// TIA Portal V21 program export: 3 tag tables, 4 data types, 7 data blocks, 12 code blocks (in call order from the OBs), 2 instance data blocks

VAR_GLOBAL   // PLC tag table "DIAG"
   D_Supply_MOD2 AT %I200.0 : Bool;   //    {ExternalWritable false}
   D_Supply_MOD3 AT %I200.1 : Bool;   //    {ExternalWritable false}
   D_Supply_MOD4 AT %I200.2 : Bool;   //    {ExternalWritable false}
   D_Supply_MOD5 AT %I200.3 : Bool;   //    {ExternalWritable false}
   D_Reserve_200_4 AT %I200.4 : Bool;   //    {ExternalWritable false}
   D_Reserve_200_5 AT %I200.5 : Bool;   //    {ExternalWritable false}
   D_Reserve_200_6 AT %I200.6 : Bool;   //    {ExternalWritable false}
   D_Reserve_200_7 AT %I200.7 : Bool;   //    {ExternalWritable false}
   D_Reserve_201_0 AT %I201.0 : Bool;   //    {ExternalWritable false}
   D_Reserve_201_1 AT %I201.1 : Bool;   //    {ExternalWritable false}
   D_Reserve_201_2 AT %I201.2 : Bool;   //    {ExternalWritable false}
   D_Reserve_201_3 AT %I201.3 : Bool;   //    {ExternalWritable false}
   D_Reserve_201_4 AT %I201.4 : Bool;   //    {ExternalWritable false}
   D_Reserve_201_5 AT %I201.5 : Bool;   //    {ExternalWritable false}
   D_Reserve_201_6 AT %I201.6 : Bool;   //    {ExternalWritable false}
   D_Reserve_201_7 AT %I201.7 : Bool;   //    {ExternalWritable false}
   D_Reserve_202_0 AT %I202.0 : Bool;   //    {ExternalWritable false}
   D_Reserve_202_1 AT %I202.1 : Bool;   //    {ExternalWritable false}
   D_Reserve_202_2 AT %I202.2 : Bool;   //    {ExternalWritable false}
   D_Reserve_202_3 AT %I202.3 : Bool;   //    {ExternalWritable false}
   D_Reserve_202_4 AT %I202.4 : Bool;   //    {ExternalWritable false}
   D_Reserve_202_5 AT %I202.5 : Bool;   //    {ExternalWritable false}
   D_Reserve_202_6 AT %I202.6 : Bool;   //    {ExternalWritable false}
   D_Reserve_202_7 AT %I202.7 : Bool;   //    {ExternalWritable false}
   D_Reserve_203_0 AT %I203.0 : Bool;   //    {ExternalWritable false}
   D_Reserve_203_1 AT %I203.1 : Bool;   //    {ExternalWritable false}
   D_Reserve_203_2 AT %I203.2 : Bool;   //    {ExternalWritable false}
   D_Reserve_203_3 AT %I203.3 : Bool;   //    {ExternalWritable false}
   D_Reserve_203_4 AT %I203.4 : Bool;   //    {ExternalWritable false}
   D_Reserve_203_5 AT %I203.5 : Bool;   //    {ExternalWritable false}
   D_Reserve_203_6 AT %I203.6 : Bool;   //    {ExternalWritable false}
   D_Reserve_203_7 AT %I203.7 : Bool;   //    {ExternalWritable false}
   D_Feedback_MOD2 AT %I204.0 : Bool;   //    {ExternalWritable false}
   D_Feedback_MOD3 AT %I204.1 : Bool;   //    {ExternalWritable false}
   D_Feedback_MOD4 AT %I204.2 : Bool;   //    {ExternalWritable false}
   D_Feedback_MOD5 AT %I204.3 : Bool;   //    {ExternalWritable false}
   D_Reserve_204_4 AT %I204.4 : Bool;   //    {ExternalWritable false}
   D_Reserve_204_5 AT %I204.5 : Bool;   //    {ExternalWritable false}
   D_Reserve_204_6 AT %I204.6 : Bool;   //    {ExternalWritable false}
   D_Reserve_204_7 AT %I204.7 : Bool;   //    {ExternalWritable false}
   D_Reserve_205_0 AT %I205.0 : Bool;   //    {ExternalWritable false}
   D_Reserve_205_1 AT %I205.1 : Bool;   //    {ExternalWritable false}
   D_Reserve_205_2 AT %I205.2 : Bool;   //    {ExternalWritable false}
   D_Reserve_205_3 AT %I205.3 : Bool;   //    {ExternalWritable false}
   D_Reserve_205_4 AT %I205.4 : Bool;   //    {ExternalWritable false}
   D_Reserve_205_5 AT %I205.5 : Bool;   //    {ExternalWritable false}
   D_Reserve_205_6 AT %I205.6 : Bool;   //    {ExternalWritable false}
   D_Reserve_205_7 AT %I205.7 : Bool;   //    {ExternalWritable false}
END_VAR

VAR_GLOBAL   // PLC tag table "Default tag table"
   System_Byte AT %MB1 : Byte;
   FirstScan AT %M1.0 : Bool;
   DiagStatusUpdate AT %M1.1 : Bool;
   AlwaysTRUE AT %M1.2 : Bool;
   AlwaysFALSE AT %M1.3 : Bool;
   Clock_Byte AT %MB0 : Byte;
   Clock_10Hz AT %M0.0 : Bool;
   Clock_5Hz AT %M0.1 : Bool;
   "Clock_2.5Hz" AT %M0.2 : Bool;
   Clock_2Hz AT %M0.3 : Bool;
   "Clock_1.25Hz" AT %M0.4 : Bool;
   Clock_1Hz AT %M0.5 : Bool;
   "Clock_0.625Hz" AT %M0.6 : Bool;
   "Clock_0.5Hz" AT %M0.7 : Bool;
END_VAR

VAR_GLOBAL   // PLC tag table "Standard-Variablentabelle"
   "High sensor" AT %I0.0 : Bool;
   "Low sensor" AT %I0.1 : Bool;
   "Pallet sensor" AT %I0.2 : Bool;
   Loaded AT %I0.3 : Bool;
   "At left entry" AT %I0.4 : Bool;
   "At left exit" AT %I0.5 : Bool;
   "At right entry" AT %I0.6 : Bool;
   "At right exit" AT %I0.7 : Bool;
   Start AT %I1.0 : Bool;
   Reset AT %I1.1 : Bool;
   Stop AT %I1.2 : Bool;
   "Emergency stop" AT %I1.3 : Bool;
   Auto AT %I1.4 : Bool;
   Running AT %I1.5 : Bool;
   "Conveyor entry" AT %Q0.0 : Bool;
   Load AT %Q0.1 : Bool;
   Unload AT %Q0.2 : Bool;
   "Trans left" AT %Q0.3 : Bool;
   "Trans right" AT %Q0.4 : Bool;
   "Conveyor left" AT %Q0.5 : Bool;
   "Conveyor right" AT %Q0.6 : Bool;
   "Start light" AT %Q0.7 : Bool;
   "Reset light" AT %Q1.0 : Bool;
   "Stop light" AT %Q1.1 : Bool;
   "Counter" AT %QW30 : Int;
END_VAR

TYPE "UDT_ Caja"
   STRUCT
      Alta : Bool;
      Baja : Bool;
   END_STRUCT;
END_TYPE

TYPE "UDT_Contador"
   STRUCT
      Total : Int;
      Altas : Int;
      Bajas : Int;
   END_STRUCT;
END_TYPE

TYPE "UDT_Settings"
   STRUCT
      AlarmDelays : Struct
         Protection : Time;
         Communication : Time;
         DriveFault : Time;
         LowCurrent : Time;
         WorkConfirmation : Time;
         Tank : Time := T#5m;
         Sensor { ExternalAccessible := 'False'; ExternalVisible := 'False'; ExternalWritable := 'False'} : Time;
      END_STRUCT;
      Sensors : Struct
         LiquidLevel : Struct
            Tank_1 : "AnalogInputSettings";
            Tank_2 : "AnalogInputSettings";
         END_STRUCT;
      END_STRUCT;
   END_STRUCT;
END_TYPE

TYPE "UDT_WORK_CNT"
   STRUCT
      S : USInt;
      "M" : USInt;
      H : UDInt;
   END_STRUCT;
END_TYPE

DATA_BLOCK "DB_Celda"   // DB1
{ S7_Optimized_Access := 'TRUE' }
// stored: MemoryReserve 100
   VAR
      Caja : "UDT_ Caja";
      Contador { S7_SetPoint := 'True'} : "UDT_Contador";
      "Sistema en marcha" { S7_SetPoint := 'True'} : Bool;
      "Modo auto" { S7_SetPoint := 'True'} : Bool;
      Emergencia { S7_SetPoint := 'True'} : Bool;
      Clasificando { S7_SetPoint := 'True'} : Bool;
   END_VAR
BEGIN
END_DATA_BLOCK

DATA_BLOCK "Simulation_DB"   // DB2
{ S7_Optimized_Access := 'TRUE'; DB_Accessible_From_OPC_UA := 'FALSE' }
// stored: AutoNumber false, DBAccessibleFromOPCUA false, DBAccessibleFromWebserver false, MemoryReserve 100
   VAR
      Simulation { ExternalAccessible := 'False'; ExternalVisible := 'False'; ExternalWritable := 'False'} : Bool;
      DigitalInputs : Struct
         EmergencyStop : Bool;
         Start : Bool;
         Stop : Bool;
         Reset : Bool;
         ContactorON : Array[1..2] of Bool;
         SoftstartON : Array[1..2] of Bool;
         SoftstartBypassed : Array[1..2] of Bool;
         SoftstartFault : Array[1..2] of Bool;
         Protection : Array[1..2] of Bool;
      END_STRUCT;
      TankLevel { ExternalWritable := 'False'} : Array[1..2] of Int;
   END_VAR
BEGIN
END_DATA_BLOCK

DATA_BLOCK "InputValues_DB"   // DB101
{ S7_Optimized_Access := 'TRUE'; DB_Accessible_From_OPC_UA := 'FALSE' }
// stored: AutoNumber false, DBAccessibleFromOPCUA false, DBAccessibleFromWebserver false, MemoryReserve 100
   VAR
      InputsDigital { ExternalWritable := 'False'} : Struct
         EmergencyStop { ExternalAccessible := 'False'; ExternalVisible := 'False'} : Bool;
         Start : Bool;
         Stop : Bool;
         Reset : Bool;
         ContactorON : Array[1..2] of Bool;
         SoftstartON : Array[1..2] of Bool;
         SoftstartBypassed : Array[1..2] of Bool;
         SoftstartFault : Array[1..2] of Bool;
         Protection : Array[1..2] of Bool;
      END_STRUCT;
      TankLevel { ExternalWritable := 'False'} : Array[1..2] of Real;
   END_VAR
BEGIN
END_DATA_BLOCK

DATA_BLOCK "AlarmsLogic_DB"   // DB202
{ S7_Optimized_Access := 'TRUE'; DB_Accessible_From_OPC_UA := 'FALSE' }
// stored: AutoNumber false, DBAccessibleFromOPCUA false, DBAccessibleFromWebserver false, MemoryReserve 100
BEGIN
END_DATA_BLOCK

DATA_BLOCK "Alarms_DB"   // DB201
{ S7_Optimized_Access := 'FALSE'; DB_Accessible_From_OPC_UA := 'FALSE' }
// stored: AutoNumber false, DBAccessibleFromOPCUA false, DBAccessibleFromWebserver false
   VAR
      General { ExternalWritable := 'False'} : Struct
         EmergencyStop : Bool;
      END_STRUCT;
      PLC { ExternalWritable := 'False'} : Struct
         SupplyModule2 : Bool;
         SupplyModule3 : Bool;
         SupplyModule4 : Bool;
         SupplyModule5 : Bool;
         FeedbackModule2 : Bool;
         FeedbackModule3 : Bool;
         FeedbackModule4 : Bool;
         FeedbackModule5 : Bool;
      END_STRUCT;
      Sensors { ExternalWritable := 'False'} : Struct
         TankLevel1_Wiring : Bool;
         TankLevel2_Wiring : Bool;
      END_STRUCT;
      Pumps { ExternalWritable := 'False'} : Struct
         CircuitProtection_1 : Bool;
         ContactorNotON_1 : Bool;
         ContactorNotOFF_1 : Bool;
         SoftstartNotON_1 : Bool;
         SoftstartNotBypassed_1 : Bool;
         SoftstartStuckBypassed_1 : Bool;
         SoftstartNotOFF_1 : Bool;
         SoftstartFault_1 : Bool;
         CircuitProtection_2 : Bool;
         ContactorNotON_2 : Bool;
         ContactorNotOFF_2 : Bool;
         SoftstartNotON_2 : Bool;
         SoftstartNotBypassed_2 : Bool;
         SoftstartStuckBypassed_2 : Bool;
         SoftstartNotOFF_2 : Bool;
         SoftstartFault_2 : Bool;
      END_STRUCT;
   END_VAR
BEGIN
END_DATA_BLOCK

DATA_BLOCK "HMI_Counters_DB"   // DB701
{ S7_Optimized_Access := 'TRUE' }
// stored: AutoNumber false, DBAccessibleFromWebserver false, MemoryReserve 100
   VAR
      ResetCounters { ExternalAccessible := 'False'; ExternalVisible := 'False'; ExternalWritable := 'False'} : Bool;
   END_VAR
   VAR RETAIN
      Machine : "UDT_WORK_CNT";
      Pump : Array[1..2] of "UDT_WORK_CNT";
   END_VAR
BEGIN
END_DATA_BLOCK

DATA_BLOCK "HMI_DB"   // DB700
{ S7_Optimized_Access := 'TRUE' }
// stored: AutoNumber false, DBAccessibleFromWebserver false, MemoryReserve 100
   VAR
      MachineState { ExternalWritable := 'False'} : USInt;
      Device { ExternalAccessible := 'False'; ExternalVisible := 'False'; ExternalWritable := 'False'} : Struct
         Pump : Array[1..2] of "UDT_Device";
      END_STRUCT;
      Devices_Status { ExternalWritable := 'False'} : Struct
         Pump : Array[1..2] of Int;
      END_STRUCT;
   END_VAR
BEGIN
END_DATA_BLOCK

ORGANIZATION_BLOCK "Main"   // OB1, LAD, ProgramCycle
TITLE = Main loop
{ S7_Optimized_Access := 'TRUE' }
// stored: SetENOAutomatically false
   VAR_INPUT
      Initial_Call : Bool;
      Remanence : Bool;
   END_VAR
BEGIN

REGION Network 1: Konnektierungsbaustein für PLC-Lab
   // #Deutsch (#English below)
   // Im Netzwerk 1 wird der Konnektierungsbaustein für PLC-Lab aufgerufen.
   // Dieser Aufruf darf nicht entfernt werden!
   // 
   // #English
   // The connection block for PLC-Lab is called up in network 1.
   // This call must not be removed!
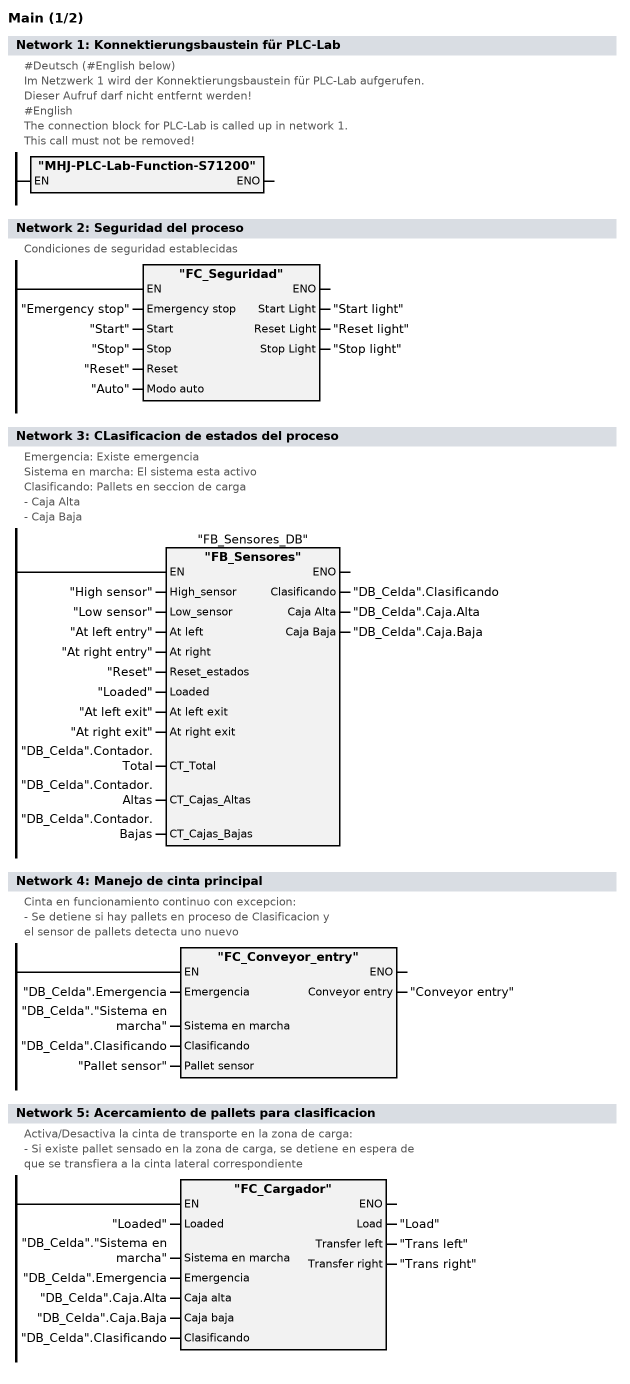
   RUNG wire#powerrail
      "MHJ-PLC-Lab-Function-S71200"()
   END_RUNG
   // the same network as SCL:
   "MHJ-PLC-Lab-Function-S71200"();
END_REGION

REGION Network 2: Seguridad del proceso
   // Condiciones de seguridad establecidas
   RUNG wire#powerrail
      "FC_Seguridad"("Emergency stop" := "Emergency stop", Start := "Start", Stop := "Stop", Reset := "Reset", "Modo auto" := "Auto", "Start Light" => "Start light", "Reset Light" => "Reset light", "Stop Light" => "Stop light")
   END_RUNG
   // the same network as SCL:
   "FC_Seguridad"("Emergency stop" := "Emergency stop",
                  Start := "Start",
                  Stop := "Stop",
                  Reset := "Reset",
                  "Modo auto" := "Auto",
                  "Start Light" => "Start light",
                  "Reset Light" => "Reset light",
                  "Stop Light" => "Stop light");
END_REGION

REGION Network 3: CLasificacion de estados del proceso
   // Emergencia: Existe emergencia
   // Sistema en marcha: El sistema esta activo
   // Clasificando: Pallets en seccion de carga
   // - Caja Alta
   // - Caja Baja
   RUNG wire#powerrail
      "FB_Sensores_DB"(High_sensor := "High sensor", Low_sensor := "Low sensor", "At left" := "At left entry", "At right" := "At right entry", Reset_estados := "Reset", Loaded := "Loaded", "At left exit" := "At left exit", "At right exit" := "At right exit", CT_Total := "DB_Celda".Contador.Total, CT_Cajas_Altas := "DB_Celda".Contador.Altas, CT_Cajas_Bajas := "DB_Celda".Contador.Bajas, Clasificando => "DB_Celda".Clasificando, "Caja Alta" => "DB_Celda".Caja.Alta, "Caja Baja" => "DB_Celda".Caja.Baja)
   END_RUNG
   // the same network as SCL:
   "FB_Sensores_DB"(High_sensor := "High sensor",   // "FB_Sensores"
                    Low_sensor := "Low sensor",
                    "At left" := "At left entry",
                    "At right" := "At right entry",
                    Reset_estados := "Reset",
                    Loaded := "Loaded",
                    "At left exit" := "At left exit",
                    "At right exit" := "At right exit",
                    CT_Total := "DB_Celda".Contador.Total,
                    CT_Cajas_Altas := "DB_Celda".Contador.Altas,
                    CT_Cajas_Bajas := "DB_Celda".Contador.Bajas,
                    Clasificando => "DB_Celda".Clasificando,
                    "Caja Alta" => "DB_Celda".Caja.Alta,
                    "Caja Baja" => "DB_Celda".Caja.Baja);
END_REGION

REGION Network 4: Manejo de cinta principal
   // Cinta en funcionamiento continuo con excepcion:
   // - Se detiene si hay pallets en proceso de Clasificacion y 
   //   el sensor de pallets detecta uno nuevo
   RUNG wire#powerrail
      "FC_Conveyor_entry"(Emergencia := "DB_Celda".Emergencia, "Sistema en marcha" := "DB_Celda"."Sistema en marcha", Clasificando := "DB_Celda".Clasificando, "Pallet sensor" := "Pallet sensor", "Conveyor entry" => "Conveyor entry")
   END_RUNG
   // the same network as SCL:
   "FC_Conveyor_entry"(Emergencia := "DB_Celda".Emergencia,
                       "Sistema en marcha" := "DB_Celda"."Sistema en marcha",
                       Clasificando := "DB_Celda".Clasificando,
                       "Pallet sensor" := "Pallet sensor",
                       "Conveyor entry" => "Conveyor entry");
END_REGION

REGION Network 5: Acercamiento de pallets para clasificacion
   // Activa/Desactiva la cinta de transporte en la zona de carga:
   // - Si existe pallet sensado en la zona de carga, se detiene en espera de
   //   que se transfiera a la cinta lateral correspondiente
   RUNG wire#powerrail
      "FC_Cargador"(Loaded := "Loaded", "Sistema en marcha" := "DB_Celda"."Sistema en marcha", Emergencia := "DB_Celda".Emergencia, "Caja alta" := "DB_Celda".Caja.Alta, "Caja baja" := "DB_Celda".Caja.Baja, Clasificando := "DB_Celda".Clasificando, Load => "Load", "Transfer left" => "Trans left", "Transfer right" => "Trans right")
   END_RUNG
   // the same network as SCL:
   "FC_Cargador"(Loaded := "Loaded",
                 "Sistema en marcha" := "DB_Celda"."Sistema en marcha",
                 Emergencia := "DB_Celda".Emergencia,
                 "Caja alta" := "DB_Celda".Caja.Alta,
                 "Caja baja" := "DB_Celda".Caja.Baja,
                 Clasificando := "DB_Celda".Clasificando,
                 Load => "Load",
                 "Transfer left" => "Trans left",
                 "Transfer right" => "Trans right");
END_REGION

REGION Network 6: Manejo de Cintas Laterales
   // Siempre activas si el sistema esta en marcha
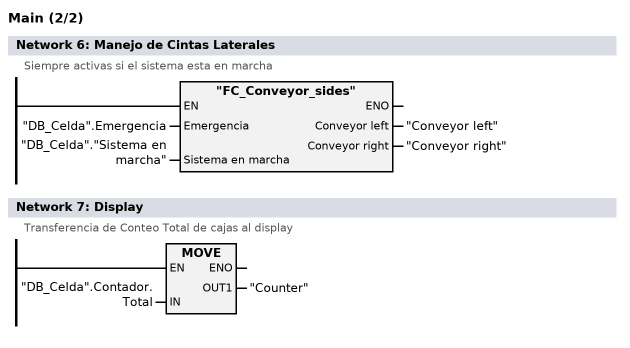
   RUNG wire#powerrail
      "FC_Conveyor_sides"(Emergencia := "DB_Celda".Emergencia, "Sistema en marcha" := "DB_Celda"."Sistema en marcha", "Conveyor left" => "Conveyor left", "Conveyor right" => "Conveyor right")
   END_RUNG
   // the same network as SCL:
   "FC_Conveyor_sides"(Emergencia := "DB_Celda".Emergencia,
                       "Sistema en marcha" := "DB_Celda"."Sistema en marcha",
                       "Conveyor left" => "Conveyor left",
                       "Conveyor right" => "Conveyor right");
END_REGION

REGION Network 7: Display
   // Transferencia de Conteo Total de cajas al display
   RUNG wire#powerrail
      Move(in := "DB_Celda".Contador.Total, out1 => "Counter")
   END_RUNG
   // the same network as SCL:
   "Counter" := "DB_Celda".Contador.Total;
END_REGION
END_ORGANIZATION_BLOCK

FUNCTION "MHJ-PLC-Lab-Function-S71200" : Void   // FC9000, SCL
{ S7_Optimized_Access := 'TRUE' }
// stored: AutoNumber false, SetENOAutomatically false
   VAR_TEMP
      rdTimeReturn : Int;
      outputTime : DTL;
      SyncVal : Byte;
      forVal : Int;
      forVal_2 : Int;
      Value : Byte;
   END_VAR
   VAR CONSTANT
      CompVal : Byte := 16#34;
      Value_01 : Byte := 16#11;
      Value_01_DW : DWord := 16#A165_D992;
      Value_02_DW : DWord := 16#58BE_4401;
   END_VAR
BEGIN

   #Value:=PEEK(area := 16#82,
        dbNumber := 0,
        byteOffset := 511);
   #Value := #Value + 1;

   POKE(area := 16#82,
        dbNumber := 0,
        byteOffset := 511,
        value := #Value);

   POKE(area:=16#81,
        dbNumber:=0,
        byteOffset:=1016,
        value:=#Value_01_DW);
   POKE(area := 16#81,
        dbNumber := 0,
        byteOffset := 1020,
        value := #Value_02_DW);

   POKE(area := 16#81,
        dbNumber := 0,
        byteOffset := 511,
        value := B#16#00);

   For #forVal := 0 To 120 Do
       For #forVal_2:=0 To 10 Do
           #rdTimeReturn:=RD_SYS_T(#outputTime);
           #rdTimeReturn := WR_SYS_T(#outputTime);
           #rdTimeReturn := RD_SYS_T(#outputTime);
           #rdTimeReturn := WR_SYS_T(#outputTime);
       End_For;
       #SyncVal:= PEEK(area := 16#81,
                      dbNumber := 0,
                      byteOffset := 511);
       If #SyncVal = #CompVal Then
          Goto M_1;
       End_If;
   End_For;
   Return;

   M_1:
   POKE(area := 16#81,
        dbNumber := 0,
        byteOffset := 511,
        value := B#16#0);
END_FUNCTION

FUNCTION "FC_Seguridad" : Void   // FC1, FBD
TITLE = Funcion de seguridad
{ S7_Optimized_Access := 'TRUE' }
// stored: SetENOAutomatically false
   VAR_INPUT
      "Emergency stop" : Bool;
      Start : Bool;
      Stop : Bool;
      Reset : Bool;
      "Modo auto" : Bool;
   END_VAR
   VAR_OUTPUT
      "Start Light" : Bool;
      "Reset Light" : Bool;
      "Stop Light" : Bool;
   END_VAR
BEGIN

REGION Network 1: Aviso de emergencia
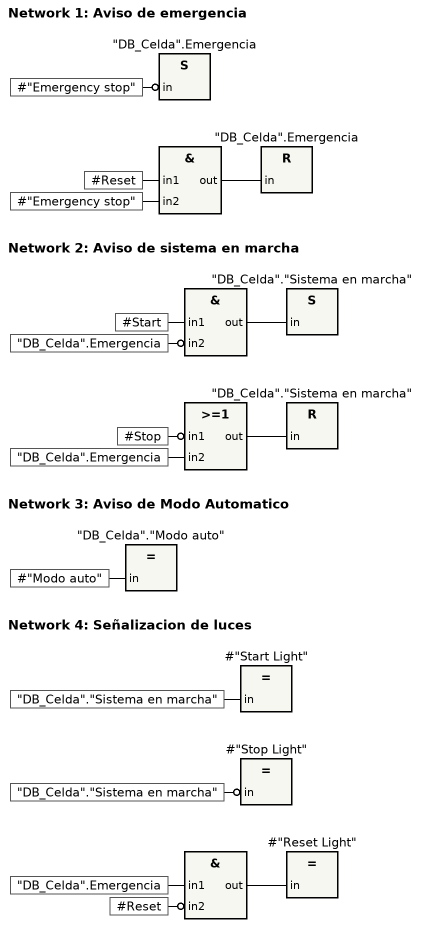
   IF NOT #"Emergency stop" THEN "DB_Celda".Emergencia := TRUE; END_IF;
   IF #Reset AND #"Emergency stop" THEN "DB_Celda".Emergencia := FALSE; END_IF;
END_REGION

REGION Network 2: Aviso de sistema en marcha
   IF #Start AND NOT "DB_Celda".Emergencia THEN "DB_Celda"."Sistema en marcha" := TRUE; END_IF;
   IF NOT #Stop OR "DB_Celda".Emergencia THEN "DB_Celda"."Sistema en marcha" := FALSE; END_IF;
END_REGION

REGION Network 3: Aviso de Modo Automatico
   "DB_Celda"."Modo auto" := #"Modo auto";
END_REGION

REGION Network 4: Señalizacion de luces
   #"Start Light" := "DB_Celda"."Sistema en marcha";
   #"Stop Light" := NOT "DB_Celda"."Sistema en marcha";
   #"Reset Light" := "DB_Celda".Emergencia AND NOT #Reset;
END_REGION
END_FUNCTION

FUNCTION_BLOCK "FB_Sensores"   // FB1, LAD
TITLE = Asignacion de estados del proceso
{ S7_Optimized_Access := 'TRUE' }
// stored: MemoryReserve 100, SetENOAutomatically false
   VAR_INPUT
      High_sensor : Bool;
      Low_sensor : Bool;
      "At left" : Bool;
      "At right" : Bool;
      Reset_estados : Bool;
      Loaded : Bool;
      "At left exit" : Bool;
      "At right exit" : Bool;
   END_VAR
   VAR_OUTPUT
      Clasificando : Bool;
      "Caja Alta" : Bool;
      "Caja Baja" : Bool;
   END_VAR
   VAR_IN_OUT
      CT_Total : Int;
      CT_Cajas_Altas : Int;
      CT_Cajas_Bajas : Int;
   END_VAR
   VAR
      Mem_At_left : Bool;
      Mem_At_right : Bool;
      Mem_clasificando : Bool;
      Mem_At_left_exit : Bool;
      Mem_At_right_exit : Bool;
   END_VAR
   VAR_TEMP   // added for the SCL form of the ladder/FBD networks
      _w1 : Bool;
      _w2 : Bool;
   END_VAR
BEGIN

REGION Network 1: Estado: Clasificando
   // Inicio: Pallet llega a sensor de carga "Loaded"
   // Fin: Pallet sale de sensores de inicio laterales (At_Left/Right_Entry)
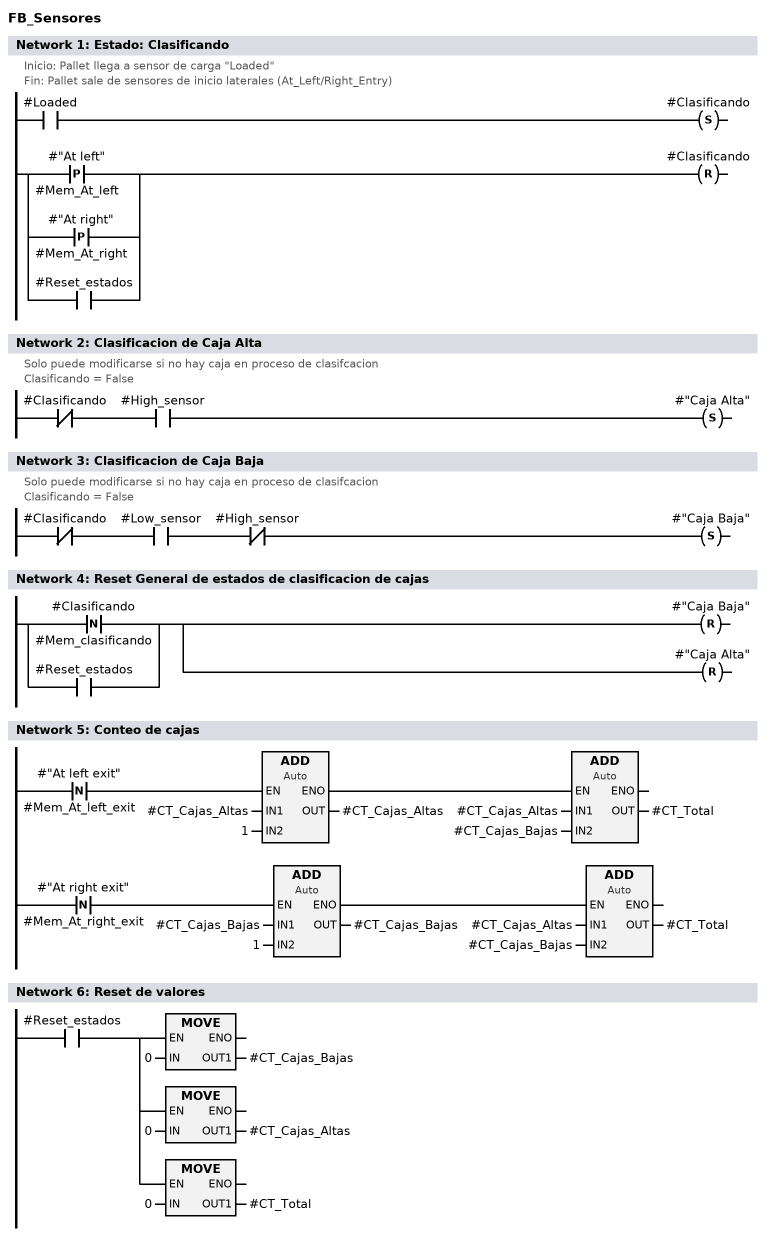
   RUNG wire#powerrail
      Contact( #Loaded )
      S_Coil( #Clasificando )
   END_RUNG
   RUNG wire#powerrail
      P_Contact(operand := #"At left", bit := #Mem_At_left)
      wire#w1
      R_Coil( #Clasificando )
   END_RUNG
   RUNG wire#powerrail
      P_Contact(operand := #"At right", bit := #Mem_At_right)
   END_RUNG wire#w1
   RUNG wire#powerrail
      Contact( #Reset_estados )
   END_RUNG wire#w1
   // the same network as SCL:
   IF #Loaded THEN #Clasificando := TRUE; END_IF;
   #_w1 := #"At left" AND NOT #Mem_At_left;   // rising edge of #"At left"
   #Mem_At_left := #"At left";
   #_w2 := #"At right" AND NOT #Mem_At_right;   // rising edge of #"At right"
   #Mem_At_right := #"At right";
   IF #_w1 OR #_w2 OR #Reset_estados THEN #Clasificando := FALSE; END_IF;
END_REGION

REGION Network 2: Clasificacion de Caja Alta
   // Solo puede modificarse si no hay caja en proceso de clasifcacion
   // Clasificando = False
   RUNG wire#powerrail
      I_Contact( #Clasificando )
      Contact( #High_sensor )
      S_Coil( #"Caja Alta" )
   END_RUNG
   // the same network as SCL:
   IF NOT #Clasificando AND #High_sensor THEN #"Caja Alta" := TRUE; END_IF;
END_REGION

REGION Network 3: Clasificacion de Caja Baja
   // Solo puede modificarse si no hay caja en proceso de clasifcacion
   // Clasificando = False
   RUNG wire#powerrail
      I_Contact( #Clasificando )
      Contact( #Low_sensor )
      I_Contact( #High_sensor )
      S_Coil( #"Caja Baja" )
   END_RUNG
   // the same network as SCL:
   IF NOT #Clasificando AND #Low_sensor AND NOT #High_sensor THEN #"Caja Baja" := TRUE; END_IF;
END_REGION

REGION Network 4: Reset General de estados de clasificacion de cajas
   RUNG wire#powerrail
      N_Contact(operand := #Clasificando, bit := #Mem_clasificando)
      wire#w1
      R_Coil( #"Caja Baja" )
   END_RUNG
   RUNG wire#powerrail
      Contact( #Reset_estados )
   END_RUNG wire#w1
   RUNG wire#w1
      R_Coil( #"Caja Alta" )
   END_RUNG
   // the same network as SCL:
   #_w1 := NOT #Clasificando AND #Mem_clasificando;   // falling edge of #Clasificando
   #Mem_clasificando := #Clasificando;
   IF #_w1 OR #Reset_estados THEN
       #"Caja Baja" := FALSE;
       #"Caja Alta" := FALSE;
   END_IF;
END_REGION

REGION Network 5: Conteo de cajas
   RUNG wire#powerrail
      N_Contact(operand := #"At left exit", bit := #Mem_At_left_exit)
      Add(in1 := #CT_Cajas_Altas, in2 := 1, out => #CT_Cajas_Altas)
      Add(in1 := #CT_Cajas_Altas, in2 := #CT_Cajas_Bajas, out => #CT_Total)
   END_RUNG
   RUNG wire#powerrail
      N_Contact(operand := #"At right exit", bit := #Mem_At_right_exit)
      Add(in1 := #CT_Cajas_Bajas, in2 := 1, out => #CT_Cajas_Bajas)
      Add(in1 := #CT_Cajas_Altas, in2 := #CT_Cajas_Bajas, out => #CT_Total)
   END_RUNG
   // the same network as SCL:
   #_w1 := NOT #"At left exit" AND #Mem_At_left_exit;   // falling edge of #"At left exit"
   #Mem_At_left_exit := #"At left exit";
   IF #_w1 THEN
       #CT_Cajas_Altas := #CT_Cajas_Altas + 1;
       #CT_Total := #CT_Cajas_Altas + #CT_Cajas_Bajas;
   END_IF;
   #_w2 := NOT #"At right exit" AND #Mem_At_right_exit;   // falling edge of #"At right exit"
   #Mem_At_right_exit := #"At right exit";
   IF #_w2 THEN
       #CT_Cajas_Bajas := #CT_Cajas_Bajas + 1;
       #CT_Total := #CT_Cajas_Altas + #CT_Cajas_Bajas;
   END_IF;
END_REGION

REGION Network 6: Reset de valores
   RUNG wire#powerrail
      Contact( #Reset_estados )
      wire#w1
      Move(in := 0, out1 => #CT_Cajas_Bajas)
   END_RUNG
   RUNG wire#w1
      Move(in := 0, out1 => #CT_Cajas_Altas)
   END_RUNG
   RUNG wire#w1
      Move(in := 0, out1 => #CT_Total)
   END_RUNG
   // the same network as SCL:
   IF #Reset_estados THEN
       #CT_Cajas_Bajas := 0;
       #CT_Cajas_Altas := 0;
       #CT_Total := 0;
   END_IF;
END_REGION
END_FUNCTION_BLOCK

FUNCTION "FC_Conveyor_entry" : Void   // FC2, LAD
TITLE = Control de Cinta Principal
{ S7_Optimized_Access := 'TRUE' }
// stored: SetENOAutomatically false
   VAR_INPUT
      Emergencia : Bool;
      "Sistema en marcha" : Bool;
      Clasificando : Bool;
      "Pallet sensor" : Bool;
   END_VAR
   VAR_OUTPUT
      "Conveyor entry" : Bool;
   END_VAR
BEGIN

REGION Network 1: Activacion/Descativacion de cinta principal
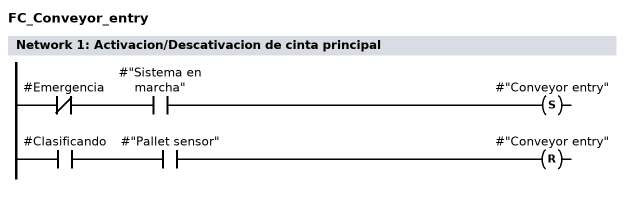
   RUNG wire#powerrail
      I_Contact( #Emergencia )
      Contact( #"Sistema en marcha" )
      S_Coil( #"Conveyor entry" )
   END_RUNG
   RUNG wire#powerrail
      Contact( #Clasificando )
      Contact( #"Pallet sensor" )
      R_Coil( #"Conveyor entry" )
   END_RUNG
   // the same network as SCL:
   IF NOT #Emergencia AND #"Sistema en marcha" THEN #"Conveyor entry" := TRUE; END_IF;
   IF #Clasificando AND #"Pallet sensor" THEN #"Conveyor entry" := FALSE; END_IF;
END_REGION
END_FUNCTION

FUNCTION "FC_Cargador" : Void   // FC3, LAD
TITLE = Sistema de carga de pallets para clasificacion
{ S7_Optimized_Access := 'TRUE' }
// stored: SetENOAutomatically false
   VAR_INPUT
      Loaded : Bool;
      "Sistema en marcha" : Bool;
      Emergencia : Bool;
      "Caja alta" : Bool;
      "Caja baja" : Bool;
      Clasificando : Bool;
   END_VAR
   VAR_OUTPUT
      Load : Bool;
      "Transfer left" : Bool;
      "Transfer right" : Bool;
   END_VAR
BEGIN

REGION Network 1: Activar/Desactivar cinta para acercamiento de pallets a sensor
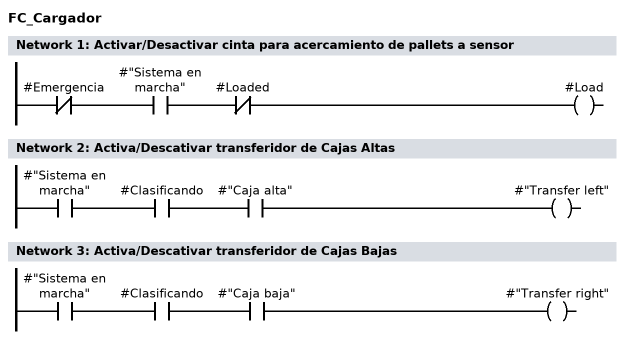
   RUNG wire#powerrail
      I_Contact( #Emergencia )
      Contact( #"Sistema en marcha" )
      I_Contact( #Loaded )
      Coil( #Load )
   END_RUNG
   // the same network as SCL:
   #Load := NOT #Emergencia AND #"Sistema en marcha" AND NOT #Loaded;
END_REGION

REGION Network 2: Activa/Descativar transferidor de Cajas Altas
   RUNG wire#powerrail
      Contact( #"Sistema en marcha" )
      Contact( #Clasificando )
      Contact( #"Caja alta" )
      Coil( #"Transfer left" )
   END_RUNG
   // the same network as SCL:
   #"Transfer left" := #"Sistema en marcha" AND #Clasificando AND #"Caja alta";
END_REGION

REGION Network 3: Activa/Descativar transferidor de Cajas Bajas
   RUNG wire#powerrail
      Contact( #"Sistema en marcha" )
      Contact( #Clasificando )
      Contact( #"Caja baja" )
      Coil( #"Transfer right" )
   END_RUNG
   // the same network as SCL:
   #"Transfer right" := #"Sistema en marcha" AND #Clasificando AND #"Caja baja";
END_REGION
END_FUNCTION

FUNCTION "FC_Conveyor_sides" : Void   // FC4, LAD
TITLE = Control de Cintas Laterales
{ S7_Optimized_Access := 'TRUE' }
// stored: SetENOAutomatically false
   VAR_INPUT
      Emergencia : Bool;
      "Sistema en marcha" : Bool;
   END_VAR
   VAR_OUTPUT
      "Conveyor left" : Bool;
      "Conveyor right" : Bool;
   END_VAR
BEGIN

REGION Network 1: Activacion/Desactivacion de cintas laterales
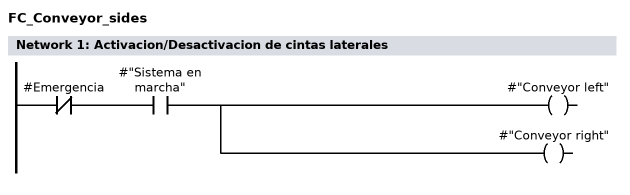
   RUNG wire#powerrail
      I_Contact( #Emergencia )
      Contact( #"Sistema en marcha" )
      wire#w1
      Coil( #"Conveyor left" )
   END_RUNG
   RUNG wire#w1
      Coil( #"Conveyor right" )
   END_RUNG
   // the same network as SCL:
   #"Conveyor left" := NOT #Emergencia AND #"Sistema en marcha";
   #"Conveyor right" := #"Conveyor left";
END_REGION
END_FUNCTION

FUNCTION_BLOCK "SimulationManagement"   // FB1, LAD
{ S7_Optimized_Access := 'TRUE' }
// stored: MemoryReserve 100, SetENOAutomatically false
BEGIN
END_FUNCTION_BLOCK

FUNCTION_BLOCK "Inputs_FB"   // FB100, LAD
{ S7_Optimized_Access := 'TRUE' }
// stored: AutoNumber false, MemoryReserve 100, SetENOAutomatically false
   VAR
      ResetEdge { ExternalAccessible := 'False'; ExternalVisible := 'False'; ExternalWritable := 'False'} : Bool;
      TankLevel { ExternalAccessible := 'False'; ExternalVisible := 'False'; ExternalWritable := 'False'} : Array[1..2] of "AnalogInput";
   END_VAR
   VAR_TEMP   // added for the SCL form of the ladder/FBD networks
      _w1 : Bool;
      _w2 : Bool;
   END_VAR
BEGIN

REGION Network 1: === General
END_REGION

REGION Network 2: Emergency stop
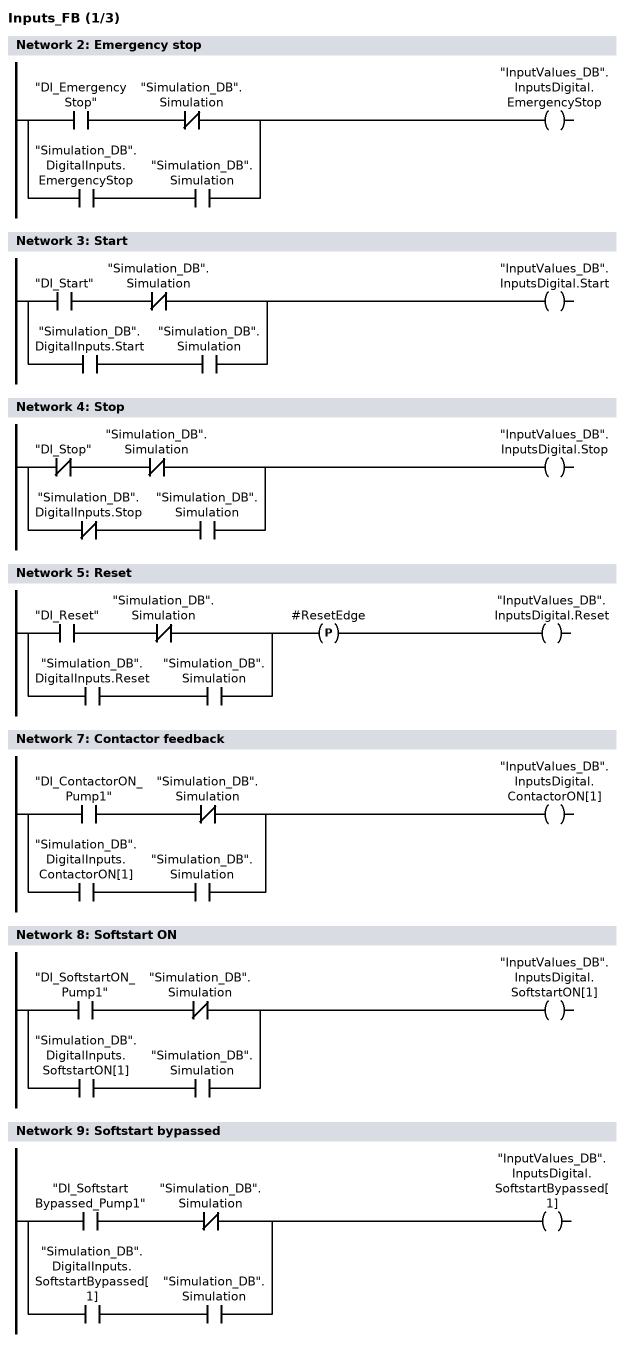
   RUNG wire#powerrail
      Contact( "DI_EmergencyStop" )
      I_Contact( "Simulation_DB".Simulation )
      wire#w1
      Coil( "InputValues_DB".InputsDigital.EmergencyStop )
   END_RUNG
   RUNG wire#powerrail
      Contact( "Simulation_DB".DigitalInputs.EmergencyStop )
      Contact( "Simulation_DB".Simulation )
   END_RUNG wire#w1
   // the same network as SCL:
   "InputValues_DB".InputsDigital.EmergencyStop := ("DI_EmergencyStop" AND NOT "Simulation_DB".Simulation) OR ("Simulation_DB".DigitalInputs.EmergencyStop AND "Simulation_DB".Simulation);
END_REGION

REGION Network 3: Start
   RUNG wire#powerrail
      Contact( "DI_Start" )
      I_Contact( "Simulation_DB".Simulation )
      wire#w1
      Coil( "InputValues_DB".InputsDigital.Start )
   END_RUNG
   RUNG wire#powerrail
      Contact( "Simulation_DB".DigitalInputs.Start )
      Contact( "Simulation_DB".Simulation )
   END_RUNG wire#w1
   // the same network as SCL:
   "InputValues_DB".InputsDigital.Start := ("DI_Start" AND NOT "Simulation_DB".Simulation) OR ("Simulation_DB".DigitalInputs.Start AND "Simulation_DB".Simulation);
END_REGION

REGION Network 4: Stop
   RUNG wire#powerrail
      I_Contact( "DI_Stop" )
      I_Contact( "Simulation_DB".Simulation )
      wire#w1
      Coil( "InputValues_DB".InputsDigital.Stop )
   END_RUNG
   RUNG wire#powerrail
      I_Contact( "Simulation_DB".DigitalInputs.Stop )
      Contact( "Simulation_DB".Simulation )
   END_RUNG wire#w1
   // the same network as SCL:
   "InputValues_DB".InputsDigital.Stop := (NOT "DI_Stop" AND NOT "Simulation_DB".Simulation) OR (NOT "Simulation_DB".DigitalInputs.Stop AND "Simulation_DB".Simulation);
END_REGION

REGION Network 5: Reset
   RUNG wire#powerrail
      Contact( "DI_Reset" )
      I_Contact( "Simulation_DB".Simulation )
      wire#w1
      P_Trig( #ResetEdge )
      Coil( "InputValues_DB".InputsDigital.Reset )
   END_RUNG
   RUNG wire#powerrail
      Contact( "Simulation_DB".DigitalInputs.Reset )
      Contact( "Simulation_DB".Simulation )
   END_RUNG wire#w1
   // the same network as SCL:
   #_w1 := ("DI_Reset" AND NOT "Simulation_DB".Simulation) OR ("Simulation_DB".DigitalInputs.Reset AND "Simulation_DB".Simulation);
   #_w2 := #_w1 AND NOT #ResetEdge;   // rising edge
   #ResetEdge := #_w1;
   "InputValues_DB".InputsDigital.Reset := #_w2;
END_REGION

REGION Network 6: === Pump 1
END_REGION

REGION Network 7: Contactor feedback
   RUNG wire#powerrail
      Contact( "DI_ContactorON_Pump1" )
      I_Contact( "Simulation_DB".Simulation )
      wire#w1
      Coil( "InputValues_DB".InputsDigital.ContactorON[1] )
   END_RUNG
   RUNG wire#powerrail
      Contact( "Simulation_DB".DigitalInputs.ContactorON[1] )
      Contact( "Simulation_DB".Simulation )
   END_RUNG wire#w1
   // the same network as SCL:
   "InputValues_DB".InputsDigital.ContactorON[1] := ("DI_ContactorON_Pump1" AND NOT "Simulation_DB".Simulation) OR ("Simulation_DB".DigitalInputs.ContactorON[1] AND "Simulation_DB".Simulation);
END_REGION

REGION Network 8: Softstart ON
   RUNG wire#powerrail
      Contact( "DI_SoftstartON_Pump1" )
      I_Contact( "Simulation_DB".Simulation )
      wire#w1
      Coil( "InputValues_DB".InputsDigital.SoftstartON[1] )
   END_RUNG
   RUNG wire#powerrail
      Contact( "Simulation_DB".DigitalInputs.SoftstartON[1] )
      Contact( "Simulation_DB".Simulation )
   END_RUNG wire#w1
   // the same network as SCL:
   "InputValues_DB".InputsDigital.SoftstartON[1] := ("DI_SoftstartON_Pump1" AND NOT "Simulation_DB".Simulation) OR ("Simulation_DB".DigitalInputs.SoftstartON[1] AND "Simulation_DB".Simulation);
END_REGION

REGION Network 9: Softstart bypassed
   RUNG wire#powerrail
      Contact( "DI_SoftstartBypassed_Pump1" )
      I_Contact( "Simulation_DB".Simulation )
      wire#w1
      Coil( "InputValues_DB".InputsDigital.SoftstartBypassed[1] )
   END_RUNG
   RUNG wire#powerrail
      Contact( "Simulation_DB".DigitalInputs.SoftstartBypassed[1] )
      Contact( "Simulation_DB".Simulation )
   END_RUNG wire#w1
   // the same network as SCL:
   "InputValues_DB".InputsDigital.SoftstartBypassed[1] := ("DI_SoftstartBypassed_Pump1" AND NOT "Simulation_DB".Simulation) OR ("Simulation_DB".DigitalInputs.SoftstartBypassed[1] AND "Simulation_DB".Simulation);
END_REGION

REGION Network 10: Softstart fault
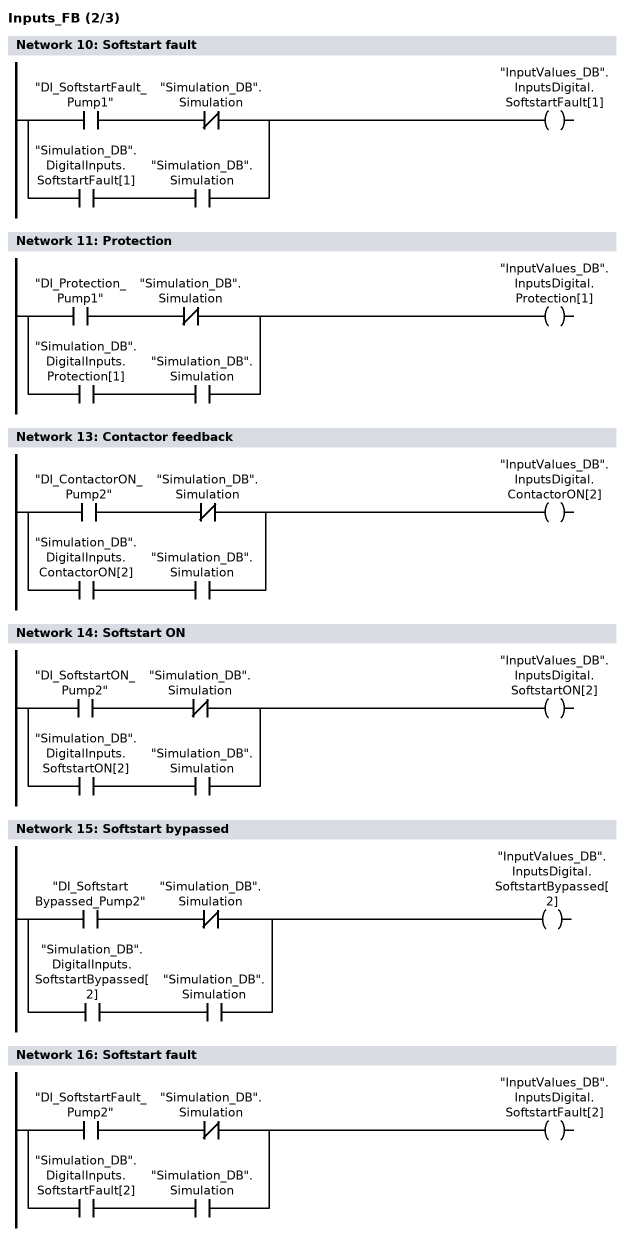
   RUNG wire#powerrail
      Contact( "DI_SoftstartFault_Pump1" )
      I_Contact( "Simulation_DB".Simulation )
      wire#w1
      Coil( "InputValues_DB".InputsDigital.SoftstartFault[1] )
   END_RUNG
   RUNG wire#powerrail
      Contact( "Simulation_DB".DigitalInputs.SoftstartFault[1] )
      Contact( "Simulation_DB".Simulation )
   END_RUNG wire#w1
   // the same network as SCL:
   "InputValues_DB".InputsDigital.SoftstartFault[1] := ("DI_SoftstartFault_Pump1" AND NOT "Simulation_DB".Simulation) OR ("Simulation_DB".DigitalInputs.SoftstartFault[1] AND "Simulation_DB".Simulation);
END_REGION

REGION Network 11: Protection
   RUNG wire#powerrail
      Contact( "DI_Protection_Pump1" )
      I_Contact( "Simulation_DB".Simulation )
      wire#w1
      Coil( "InputValues_DB".InputsDigital.Protection[1] )
   END_RUNG
   RUNG wire#powerrail
      Contact( "Simulation_DB".DigitalInputs.Protection[1] )
      Contact( "Simulation_DB".Simulation )
   END_RUNG wire#w1
   // the same network as SCL:
   "InputValues_DB".InputsDigital.Protection[1] := ("DI_Protection_Pump1" AND NOT "Simulation_DB".Simulation) OR ("Simulation_DB".DigitalInputs.Protection[1] AND "Simulation_DB".Simulation);
END_REGION

REGION Network 12: === Pump 2
END_REGION

REGION Network 13: Contactor feedback
   RUNG wire#powerrail
      Contact( "DI_ContactorON_Pump2" )
      I_Contact( "Simulation_DB".Simulation )
      wire#w1
      Coil( "InputValues_DB".InputsDigital.ContactorON[2] )
   END_RUNG
   RUNG wire#powerrail
      Contact( "Simulation_DB".DigitalInputs.ContactorON[2] )
      Contact( "Simulation_DB".Simulation )
   END_RUNG wire#w1
   // the same network as SCL:
   "InputValues_DB".InputsDigital.ContactorON[2] := ("DI_ContactorON_Pump2" AND NOT "Simulation_DB".Simulation) OR ("Simulation_DB".DigitalInputs.ContactorON[2] AND "Simulation_DB".Simulation);
END_REGION

REGION Network 14: Softstart ON
   RUNG wire#powerrail
      Contact( "DI_SoftstartON_Pump2" )
      I_Contact( "Simulation_DB".Simulation )
      wire#w1
      Coil( "InputValues_DB".InputsDigital.SoftstartON[2] )
   END_RUNG
   RUNG wire#powerrail
      Contact( "Simulation_DB".DigitalInputs.SoftstartON[2] )
      Contact( "Simulation_DB".Simulation )
   END_RUNG wire#w1
   // the same network as SCL:
   "InputValues_DB".InputsDigital.SoftstartON[2] := ("DI_SoftstartON_Pump2" AND NOT "Simulation_DB".Simulation) OR ("Simulation_DB".DigitalInputs.SoftstartON[2] AND "Simulation_DB".Simulation);
END_REGION

REGION Network 15: Softstart bypassed
   RUNG wire#powerrail
      Contact( "DI_SoftstartBypassed_Pump2" )
      I_Contact( "Simulation_DB".Simulation )
      wire#w1
      Coil( "InputValues_DB".InputsDigital.SoftstartBypassed[2] )
   END_RUNG
   RUNG wire#powerrail
      Contact( "Simulation_DB".DigitalInputs.SoftstartBypassed[2] )
      Contact( "Simulation_DB".Simulation )
   END_RUNG wire#w1
   // the same network as SCL:
   "InputValues_DB".InputsDigital.SoftstartBypassed[2] := ("DI_SoftstartBypassed_Pump2" AND NOT "Simulation_DB".Simulation) OR ("Simulation_DB".DigitalInputs.SoftstartBypassed[2] AND "Simulation_DB".Simulation);
END_REGION

REGION Network 16: Softstart fault
   RUNG wire#powerrail
      Contact( "DI_SoftstartFault_Pump2" )
      I_Contact( "Simulation_DB".Simulation )
      wire#w1
      Coil( "InputValues_DB".InputsDigital.SoftstartFault[2] )
   END_RUNG
   RUNG wire#powerrail
      Contact( "Simulation_DB".DigitalInputs.SoftstartFault[2] )
      Contact( "Simulation_DB".Simulation )
   END_RUNG wire#w1
   // the same network as SCL:
   "InputValues_DB".InputsDigital.SoftstartFault[2] := ("DI_SoftstartFault_Pump2" AND NOT "Simulation_DB".Simulation) OR ("Simulation_DB".DigitalInputs.SoftstartFault[2] AND "Simulation_DB".Simulation);
END_REGION

REGION Network 17: Protection
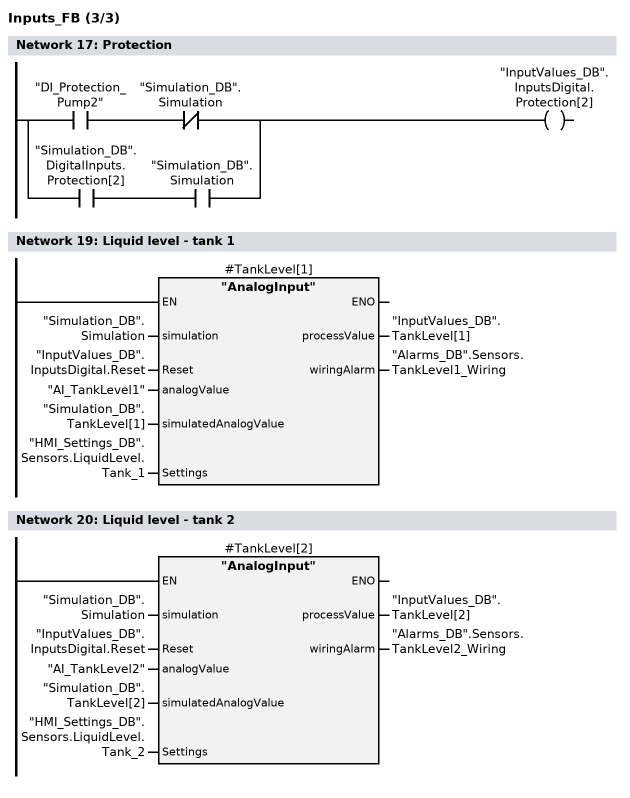
   RUNG wire#powerrail
      Contact( "DI_Protection_Pump2" )
      I_Contact( "Simulation_DB".Simulation )
      wire#w1
      Coil( "InputValues_DB".InputsDigital.Protection[2] )
   END_RUNG
   RUNG wire#powerrail
      Contact( "Simulation_DB".DigitalInputs.Protection[2] )
      Contact( "Simulation_DB".Simulation )
   END_RUNG wire#w1
   // the same network as SCL:
   "InputValues_DB".InputsDigital.Protection[2] := ("DI_Protection_Pump2" AND NOT "Simulation_DB".Simulation) OR ("Simulation_DB".DigitalInputs.Protection[2] AND "Simulation_DB".Simulation);
END_REGION

REGION Network 18: === Analog inputs
END_REGION

REGION Network 19: Liquid level - tank 1
   RUNG wire#powerrail
      #TankLevel[1](simulation := "Simulation_DB".Simulation, Reset := "InputValues_DB".InputsDigital.Reset, analogValue := "AI_TankLevel1", simulatedAnalogValue := "Simulation_DB".TankLevel[1], Settings := "HMI_Settings_DB".Sensors.LiquidLevel.Tank_1, processValue => "InputValues_DB".TankLevel[1], wiringAlarm => "Alarms_DB".Sensors.TankLevel1_Wiring)
   END_RUNG
   // the same network as SCL:
   #TankLevel[1](simulation := "Simulation_DB".Simulation,   // "AnalogInput"
                 Reset := "InputValues_DB".InputsDigital.Reset,
                 analogValue := "AI_TankLevel1",
                 simulatedAnalogValue := "Simulation_DB".TankLevel[1],
                 Settings := "HMI_Settings_DB".Sensors.LiquidLevel.Tank_1,
                 processValue => "InputValues_DB".TankLevel[1],
                 wiringAlarm => "Alarms_DB".Sensors.TankLevel1_Wiring);
END_REGION

REGION Network 20: Liquid level - tank 2
   RUNG wire#powerrail
      #TankLevel[2](simulation := "Simulation_DB".Simulation, Reset := "InputValues_DB".InputsDigital.Reset, analogValue := "AI_TankLevel2", simulatedAnalogValue := "Simulation_DB".TankLevel[2], Settings := "HMI_Settings_DB".Sensors.LiquidLevel.Tank_2, processValue => "InputValues_DB".TankLevel[2], wiringAlarm => "Alarms_DB".Sensors.TankLevel2_Wiring)
   END_RUNG
   // the same network as SCL:
   #TankLevel[2](simulation := "Simulation_DB".Simulation,   // "AnalogInput"
                 Reset := "InputValues_DB".InputsDigital.Reset,
                 analogValue := "AI_TankLevel2",
                 simulatedAnalogValue := "Simulation_DB".TankLevel[2],
                 Settings := "HMI_Settings_DB".Sensors.LiquidLevel.Tank_2,
                 processValue => "InputValues_DB".TankLevel[2],
                 wiringAlarm => "Alarms_DB".Sensors.TankLevel2_Wiring);
END_REGION
END_FUNCTION_BLOCK

FUNCTION_BLOCK "AlarmsContainer"   // FB200, LAD
{ S7_Optimized_Access := 'TRUE' }
// stored: AutoNumber false, MemoryReserve 100, SetENOAutomatically false
   VAR
      WeeklyReset { ExternalAccessible := 'False'; ExternalVisible := 'False'; ExternalWritable := 'False'} : Bool;
      MaintenanceReset : Bool;
      Edge { ExternalAccessible := 'False'; ExternalVisible := 'False'; ExternalWritable := 'False'} : Array[0..10] of Bool;
   END_VAR
   VAR_TEMP
      tempBool : Bool;
      i : USInt;
      j : USInt;
      n : DInt;
      Addr : DInt;
   END_VAR
   VAR_TEMP   // added for the SCL form of the ladder/FBD networks
      _w1 : Bool;
   END_VAR
BEGIN

REGION Network 1: ======================================= General
END_REGION

REGION Network 2: Emergency stop
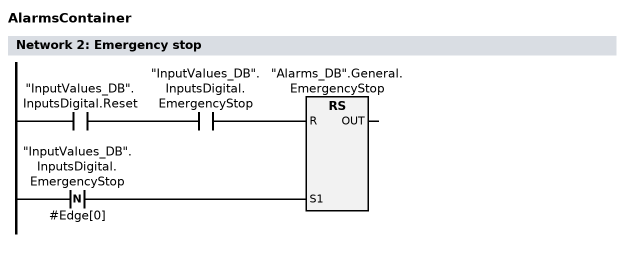
   RUNG wire#powerrail
      Contact( "InputValues_DB".InputsDigital.Reset )
      Contact( "InputValues_DB".InputsDigital.EmergencyStop )
      S_RS(operand := "Alarms_DB".General.EmergencyStop, s1 := wire#w1)
   END_RUNG
   RUNG wire#powerrail
      N_Contact(operand := "InputValues_DB".InputsDigital.EmergencyStop, bit := #Edge[0])
   END_RUNG wire#w1
   // the same network as SCL:
   #_w1 := NOT "InputValues_DB".InputsDigital.EmergencyStop AND #Edge[0];   // falling edge of "InputValues_DB".InputsDigital.EmergencyStop
   #Edge[0] := "InputValues_DB".InputsDigital.EmergencyStop;
   IF "InputValues_DB".InputsDigital.Reset AND "InputValues_DB".InputsDigital.EmergencyStop THEN
       "Alarms_DB".General.EmergencyStop := FALSE;   // RS flip-flop
   END_IF;
   IF #_w1 THEN "Alarms_DB".General.EmergencyStop := TRUE; END_IF;
END_REGION

REGION Network 3 (SCL): ======================================= PLC
   // TODO
   FOR #i := 2 TO 5 DO
       IF #i = 2 THEN
           #Addr := 200;
           #n := 0;
       ELSIF #i = 4 THEN
           #Addr := 204;
           #n := 0;
       END_IF;
       FOR #j := 0 TO 7 DO
           #tempBool := PEEK_BOOL(area := 16#81, dbNumber := 0, byteOffset := #Addr + #n, bitOffset := #j);
           IF NOT #tempBool THEN
               POKE_BOOL(area := 16#84,
                         dbNumber := 201,
                         byteOffset := #i,
                         bitOffset := #j,
                         value := TRUE);
           ELSIF "InputValues_DB".InputsDigital.Reset THEN
               POKE_BOOL(area := 16#84,
                         dbNumber := 201,
                         byteOffset := #i,
                         bitOffset := #j,
                         value := FALSE);
           END_IF;
       END_FOR;
       #n += 1;
   END_FOR;
END_REGION
END_FUNCTION_BLOCK

FUNCTION_BLOCK "MotorSoftstart"   // FB8889, LAD
{ S7_Optimized_Access := 'TRUE' }
// stored: AutoNumber false, MemoryReserve 100, SetENOAutomatically false
   VAR_INPUT
      FI_AutoConditions { ExternalAccessible := 'False'; ExternalVisible := 'False'; ExternalWritable := 'False'} : Bool;
      FI_AutoForward { ExternalAccessible := 'False'; ExternalVisible := 'False'; ExternalWritable := 'False'} : Bool;
      FI_ProfinetOK { ExternalAccessible := 'False'; ExternalVisible := 'False'; ExternalWritable := 'False'} : Bool;
      FI_CircuitProtectionOK { ExternalAccessible := 'False'; ExternalVisible := 'False'; ExternalWritable := 'False'} : Bool;
      FI_SoftstartAlarm { ExternalAccessible := 'False'; ExternalVisible := 'False'; ExternalWritable := 'False'} : Bool;
      FI_ContactorON { ExternalAccessible := 'False'; ExternalVisible := 'False'; ExternalWritable := 'False'} : Bool;
      FI_SoftstartON { ExternalAccessible := 'False'; ExternalVisible := 'False'; ExternalWritable := 'False'} : Bool;
      FI_SoftstartBypassed { ExternalAccessible := 'False'; ExternalVisible := 'False'; ExternalWritable := 'False'} : Bool;
      FI_ManualMode { ExternalAccessible := 'False'; ExternalVisible := 'False'; ExternalWritable := 'False'} : Bool;
      FI_EmergencyStop { ExternalAccessible := 'False'; ExternalVisible := 'False'; ExternalWritable := 'False'} : Bool;
      FI_Reset { ExternalAccessible := 'False'; ExternalVisible := 'False'; ExternalWritable := 'False'} : Bool;
   END_VAR
   VAR_OUTPUT
      FQ_ContactorON { ExternalAccessible := 'False'; ExternalVisible := 'False'; ExternalWritable := 'False'} : Bool;
      FQ_MotorStart { ExternalAccessible := 'False'; ExternalVisible := 'False'; ExternalWritable := 'False'} : Bool;
      FQ_AlarmCircuitProtection { ExternalAccessible := 'False'; ExternalVisible := 'False'; ExternalWritable := 'False'} : Bool;
      FQ_AlarmContactorNotON { ExternalAccessible := 'False'; ExternalVisible := 'False'; ExternalWritable := 'False'} : Bool;
      FQ_AlarmContactorNotOFF { ExternalAccessible := 'False'; ExternalVisible := 'False'; ExternalWritable := 'False'} : Bool;
      FQ_AlarmSoftstartNotON { ExternalAccessible := 'False'; ExternalVisible := 'False'; ExternalWritable := 'False'} : Bool;
      FQ_AlarmSoftstartNotBypassed { ExternalAccessible := 'False'; ExternalVisible := 'False'; ExternalWritable := 'False'} : Bool;
      FQ_AlarmSoftstartStuckBypassed { ExternalAccessible := 'False'; ExternalVisible := 'False'; ExternalWritable := 'False'} : Bool;
      FQ_AlarmSoftstartNotOFF { ExternalAccessible := 'False'; ExternalVisible := 'False'; ExternalWritable := 'False'} : Bool;
      FQ_AlarmSoftstartFault { ExternalAccessible := 'False'; ExternalVisible := 'False'; ExternalWritable := 'False'} : Bool;
   END_VAR
   VAR_IN_OUT
      FIQ_WorkTime : "UDT_WORK_CNT";
      FIQ_DeviceState : "UDT_Device";
   END_VAR
   VAR
      generalConditions { ExternalAccessible := 'False'; ExternalVisible := 'False'; ExternalWritable := 'False'} : Bool;
      Authorisation { ExternalAccessible := 'False'; ExternalVisible := 'False'; ExternalWritable := 'False'} : Bool;
      Alarm { ExternalAccessible := 'False'; ExternalVisible := 'False'; ExternalWritable := 'False'} : Bool;
      contactorON { ExternalAccessible := 'False'; ExternalVisible := 'False'; ExternalWritable := 'False'} : Bool;
      motorStart { ExternalAccessible := 'False'; ExternalVisible := 'False'; ExternalWritable := 'False'} : Bool;
      motorConfirmed { ExternalAccessible := 'False'; ExternalVisible := 'False'; ExternalWritable := 'False'} : Bool;
      Timers { ExternalAccessible := 'False'; ExternalVisible := 'False'; ExternalWritable := 'False'} : Struct
         CircuitProtection : TON_TIME;
         ContNotON : TON_TIME;
         ContNotOFF : TON_TIME;
         SoftstartNotON : TON_TIME;
         SoftstartNotOFF : TON_TIME;
         SoftstartNotBypassed : TON_TIME;
         SoftstartBypassed : TON_TIME;
         SoftstartFailure : TON_TIME;
      END_STRUCT;
      C_WORK_TIME { ExternalAccessible := 'False'; ExternalVisible := 'False'; ExternalWritable := 'False'} : "TIME_COUNTER_FB";
   END_VAR
BEGIN

REGION Network 1: General conditions
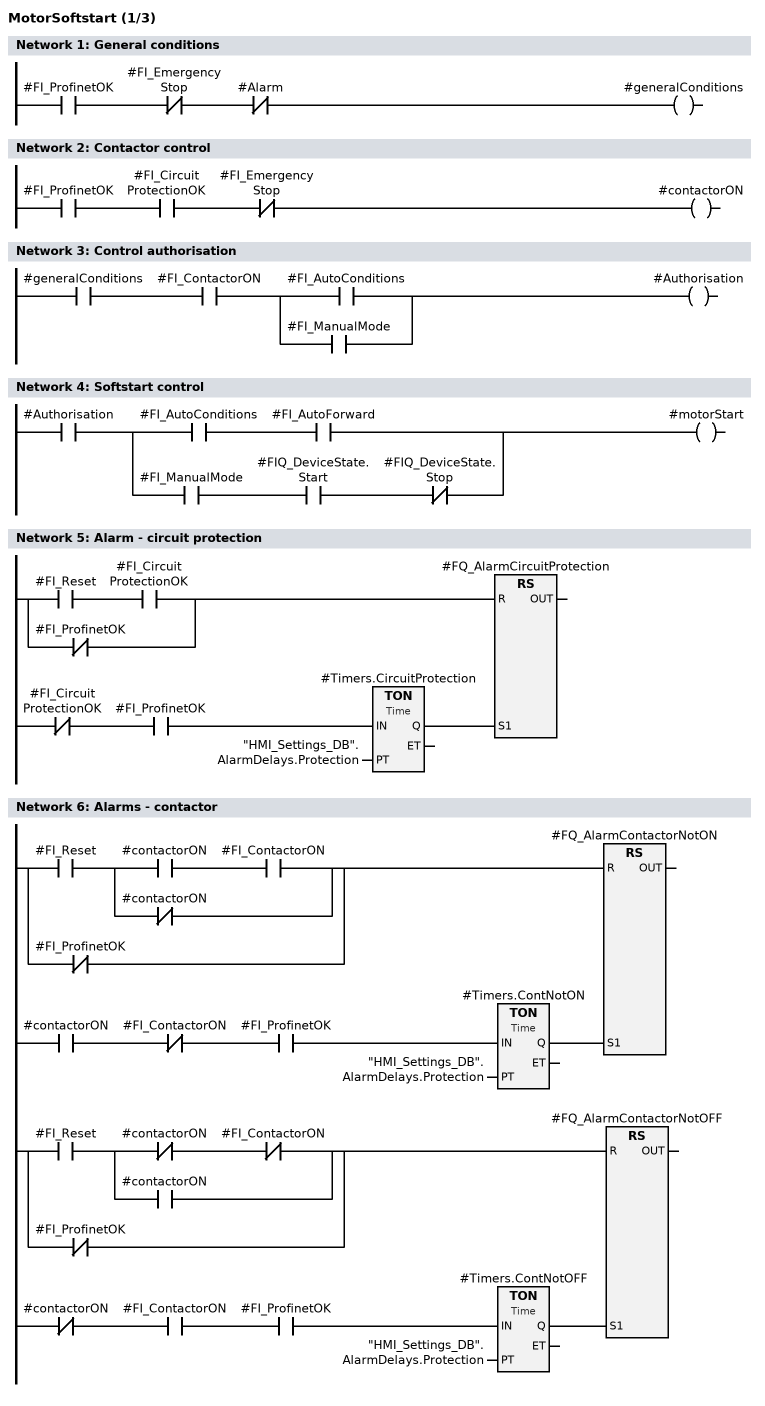
   RUNG wire#powerrail
      Contact( #FI_ProfinetOK )
      I_Contact( #FI_EmergencyStop )
      I_Contact( #Alarm )
      Coil( #generalConditions )
   END_RUNG
   // the same network as SCL:
   #generalConditions := #FI_ProfinetOK AND NOT #FI_EmergencyStop AND NOT #Alarm;
END_REGION

REGION Network 2: Contactor control
   RUNG wire#powerrail
      Contact( #FI_ProfinetOK )
      Contact( #FI_CircuitProtectionOK )
      I_Contact( #FI_EmergencyStop )
      Coil( #contactorON )
   END_RUNG
   // the same network as SCL:
   #contactorON := #FI_ProfinetOK AND #FI_CircuitProtectionOK AND NOT #FI_EmergencyStop;
END_REGION

REGION Network 3: Control authorisation
   RUNG wire#powerrail
      Contact( #generalConditions )
      Contact( #FI_ContactorON )
      wire#w1
      Contact( #FI_AutoConditions )
      wire#w2
      Coil( #Authorisation )
   END_RUNG
   RUNG wire#w1
      Contact( #FI_ManualMode )
   END_RUNG wire#w2
   // the same network as SCL:
   #Authorisation := #generalConditions AND #FI_ContactorON AND (#FI_AutoConditions OR #FI_ManualMode);
END_REGION

REGION Network 4: Softstart control
   RUNG wire#powerrail
      Contact( #Authorisation )
      wire#w1
      Contact( #FI_AutoConditions )
      Contact( #FI_AutoForward )
      wire#w2
      Coil( #motorStart )
   END_RUNG
   RUNG wire#w1
      Contact( #FI_ManualMode )
      Contact( #FIQ_DeviceState.Start )
      I_Contact( #FIQ_DeviceState.Stop )
   END_RUNG wire#w2
   // the same network as SCL:
   #motorStart := #Authorisation AND ((#FI_AutoConditions AND #FI_AutoForward) OR (#FI_ManualMode AND #FIQ_DeviceState.Start AND NOT #FIQ_DeviceState.Stop));
END_REGION

REGION Network 5: Alarm - circuit protection
   RUNG wire#powerrail
      Contact( #FI_Reset )
      Contact( #FI_CircuitProtectionOK )
      wire#w1
      S_RS(operand := #FQ_AlarmCircuitProtection, s1 := wire#w2)
   END_RUNG
   RUNG wire#powerrail
      I_Contact( #FI_ProfinetOK )
   END_RUNG wire#w1
   RUNG wire#powerrail
      I_Contact( #FI_CircuitProtectionOK )
      Contact( #FI_ProfinetOK )
      { S7_Templates := "time_type := Time" } #Timers.CircuitProtection.TON(pt := "HMI_Settings_DB".AlarmDelays.Protection, et =>)
   END_RUNG wire#w2
   // the same network as SCL:
   #Timers.CircuitProtection.TON(IN := NOT #FI_CircuitProtectionOK AND #FI_ProfinetOK,
                           PT := "HMI_Settings_DB".AlarmDelays.Protection);
   IF (#FI_Reset AND #FI_CircuitProtectionOK) OR NOT #FI_ProfinetOK THEN
       #FQ_AlarmCircuitProtection := FALSE;   // RS flip-flop
   END_IF;
   IF #Timers.CircuitProtection.Q THEN #FQ_AlarmCircuitProtection := TRUE; END_IF;
END_REGION

REGION Network 6: Alarms - contactor
   RUNG wire#powerrail
      Contact( #FI_Reset )
      wire#w1
      Contact( #contactorON )
      Contact( #FI_ContactorON )
      wire#w2
      S_RS(operand := #FQ_AlarmContactorNotON, s1 := wire#w3)
   END_RUNG
   RUNG wire#w1
      I_Contact( #contactorON )
   END_RUNG wire#w2
   RUNG wire#powerrail
      I_Contact( #FI_ProfinetOK )
   END_RUNG wire#w2
   RUNG wire#powerrail
      Contact( #contactorON )
      I_Contact( #FI_ContactorON )
      Contact( #FI_ProfinetOK )
      { S7_Templates := "time_type := Time" } #Timers.ContNotON.TON(pt := "HMI_Settings_DB".AlarmDelays.Protection, et =>)
   END_RUNG wire#w3
   RUNG wire#powerrail
      Contact( #FI_Reset )
      wire#w4
      I_Contact( #contactorON )
      I_Contact( #FI_ContactorON )
      wire#w5
      S_RS(operand := #FQ_AlarmContactorNotOFF, s1 := wire#w6)
   END_RUNG
   RUNG wire#w4
      Contact( #contactorON )
   END_RUNG wire#w5
   RUNG wire#powerrail
      I_Contact( #FI_ProfinetOK )
   END_RUNG wire#w5
   RUNG wire#powerrail
      I_Contact( #contactorON )
      Contact( #FI_ContactorON )
      Contact( #FI_ProfinetOK )
      { S7_Templates := "time_type := Time" } #Timers.ContNotOFF.TON(pt := "HMI_Settings_DB".AlarmDelays.Protection, et =>)
   END_RUNG wire#w6
   // the same network as SCL:
   #Timers.ContNotON.TON(IN := #contactorON AND NOT #FI_ContactorON AND #FI_ProfinetOK,
                         PT := "HMI_Settings_DB".AlarmDelays.Protection);
   IF (#FI_Reset AND ((#contactorON AND #FI_ContactorON) OR NOT #contactorON)) OR NOT #FI_ProfinetOK THEN
       #FQ_AlarmContactorNotON := FALSE;   // RS flip-flop
   END_IF;
   IF #Timers.ContNotON.Q THEN #FQ_AlarmContactorNotON := TRUE; END_IF;
   #Timers.ContNotOFF.TON(IN := NOT #contactorON AND #FI_ContactorON AND #FI_ProfinetOK,
                          PT := "HMI_Settings_DB".AlarmDelays.Protection);
   IF (#FI_Reset AND ((NOT #contactorON AND NOT #FI_ContactorON) OR #contactorON)) OR NOT #FI_ProfinetOK THEN
       #FQ_AlarmContactorNotOFF := FALSE;   // RS flip-flop
   END_IF;
   IF #Timers.ContNotOFF.Q THEN #FQ_AlarmContactorNotOFF := TRUE; END_IF;
END_REGION

REGION Network 7: Alarm - softstart not ON
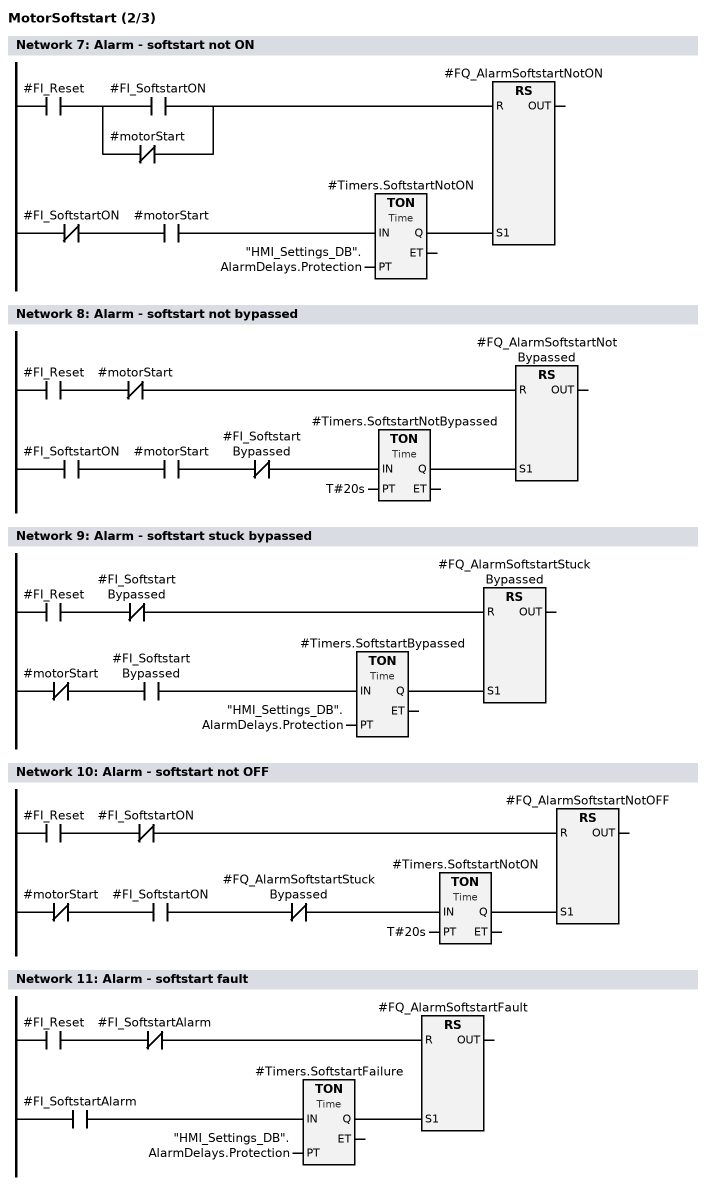
   RUNG wire#powerrail
      Contact( #FI_Reset )
      wire#w1
      Contact( #FI_SoftstartON )
      wire#w2
      S_RS(operand := #FQ_AlarmSoftstartNotON, s1 := wire#w3)
   END_RUNG
   RUNG wire#w1
      I_Contact( #motorStart )
   END_RUNG wire#w2
   RUNG wire#powerrail
      I_Contact( #FI_SoftstartON )
      Contact( #motorStart )
      { S7_Templates := "time_type := Time" } #Timers.SoftstartNotON.TON(pt := "HMI_Settings_DB".AlarmDelays.Protection, et =>)
   END_RUNG wire#w3
   // the same network as SCL:
   #Timers.SoftstartNotON.TON(IN := NOT #FI_SoftstartON AND #motorStart,
                           PT := "HMI_Settings_DB".AlarmDelays.Protection);
   IF #FI_Reset AND (#FI_SoftstartON OR NOT #motorStart) THEN
       #FQ_AlarmSoftstartNotON := FALSE;   // RS flip-flop
   END_IF;
   IF #Timers.SoftstartNotON.Q THEN #FQ_AlarmSoftstartNotON := TRUE; END_IF;
END_REGION

REGION Network 8: Alarm - softstart not bypassed
   RUNG wire#powerrail
      Contact( #FI_Reset )
      I_Contact( #motorStart )
      S_RS(operand := #FQ_AlarmSoftstartNotBypassed, s1 := wire#w1)
   END_RUNG
   RUNG wire#powerrail
      Contact( #FI_SoftstartON )
      Contact( #motorStart )
      I_Contact( #FI_SoftstartBypassed )
      { S7_Templates := "time_type := Time" } #Timers.SoftstartNotBypassed.TON(pt := T#20s, et =>)
   END_RUNG wire#w1
   // the same network as SCL:
   #Timers.SoftstartNotBypassed.TON(IN := #FI_SoftstartON AND #motorStart AND NOT #FI_SoftstartBypassed,
                           PT := T#20s);
   IF #FI_Reset AND NOT #motorStart THEN
       #FQ_AlarmSoftstartNotBypassed := FALSE;   // RS flip-flop
   END_IF;
   IF #Timers.SoftstartNotBypassed.Q THEN #FQ_AlarmSoftstartNotBypassed := TRUE; END_IF;
END_REGION

REGION Network 9: Alarm - softstart stuck bypassed
   RUNG wire#powerrail
      Contact( #FI_Reset )
      I_Contact( #FI_SoftstartBypassed )
      S_RS(operand := #FQ_AlarmSoftstartStuckBypassed, s1 := wire#w1)
   END_RUNG
   RUNG wire#powerrail
      I_Contact( #motorStart )
      Contact( #FI_SoftstartBypassed )
      { S7_Templates := "time_type := Time" } #Timers.SoftstartBypassed.TON(pt := "HMI_Settings_DB".AlarmDelays.Protection, et =>)
   END_RUNG wire#w1
   // the same network as SCL:
   #Timers.SoftstartBypassed.TON(IN := NOT #motorStart AND #FI_SoftstartBypassed,
                           PT := "HMI_Settings_DB".AlarmDelays.Protection);
   IF #FI_Reset AND NOT #FI_SoftstartBypassed THEN
       #FQ_AlarmSoftstartStuckBypassed := FALSE;   // RS flip-flop
   END_IF;
   IF #Timers.SoftstartBypassed.Q THEN #FQ_AlarmSoftstartStuckBypassed := TRUE; END_IF;
END_REGION

REGION Network 10: Alarm - softstart not OFF
   RUNG wire#powerrail
      Contact( #FI_Reset )
      I_Contact( #FI_SoftstartON )
      S_RS(operand := #FQ_AlarmSoftstartNotOFF, s1 := wire#w1)
   END_RUNG
   RUNG wire#powerrail
      I_Contact( #motorStart )
      Contact( #FI_SoftstartON )
      I_Contact( #FQ_AlarmSoftstartStuckBypassed )
      { S7_Templates := "time_type := Time" } #Timers.SoftstartNotON.TON(pt := T#20s, et =>)
   END_RUNG wire#w1
   // the same network as SCL:
   #Timers.SoftstartNotON.TON(IN := NOT #motorStart AND #FI_SoftstartON AND NOT #FQ_AlarmSoftstartStuckBypassed,
                           PT := T#20s);
   IF #FI_Reset AND NOT #FI_SoftstartON THEN
       #FQ_AlarmSoftstartNotOFF := FALSE;   // RS flip-flop
   END_IF;
   IF #Timers.SoftstartNotON.Q THEN #FQ_AlarmSoftstartNotOFF := TRUE; END_IF;
END_REGION

REGION Network 11: Alarm - softstart fault
   RUNG wire#powerrail
      Contact( #FI_Reset )
      I_Contact( #FI_SoftstartAlarm )
      S_RS(operand := #FQ_AlarmSoftstartFault, s1 := wire#w1)
   END_RUNG
   RUNG wire#powerrail
      Contact( #FI_SoftstartAlarm )
      { S7_Templates := "time_type := Time" } #Timers.SoftstartFailure.TON(pt := "HMI_Settings_DB".AlarmDelays.Protection, et =>)
   END_RUNG wire#w1
   // the same network as SCL:
   #Timers.SoftstartFailure.TON(IN := #FI_SoftstartAlarm, PT := "HMI_Settings_DB".AlarmDelays.Protection);
   IF #FI_Reset AND NOT #FI_SoftstartAlarm THEN
       #FQ_AlarmSoftstartFault := FALSE;   // RS flip-flop
   END_IF;
   IF #Timers.SoftstartFailure.Q THEN #FQ_AlarmSoftstartFault := TRUE; END_IF;
END_REGION

REGION Network 12: Any alarm
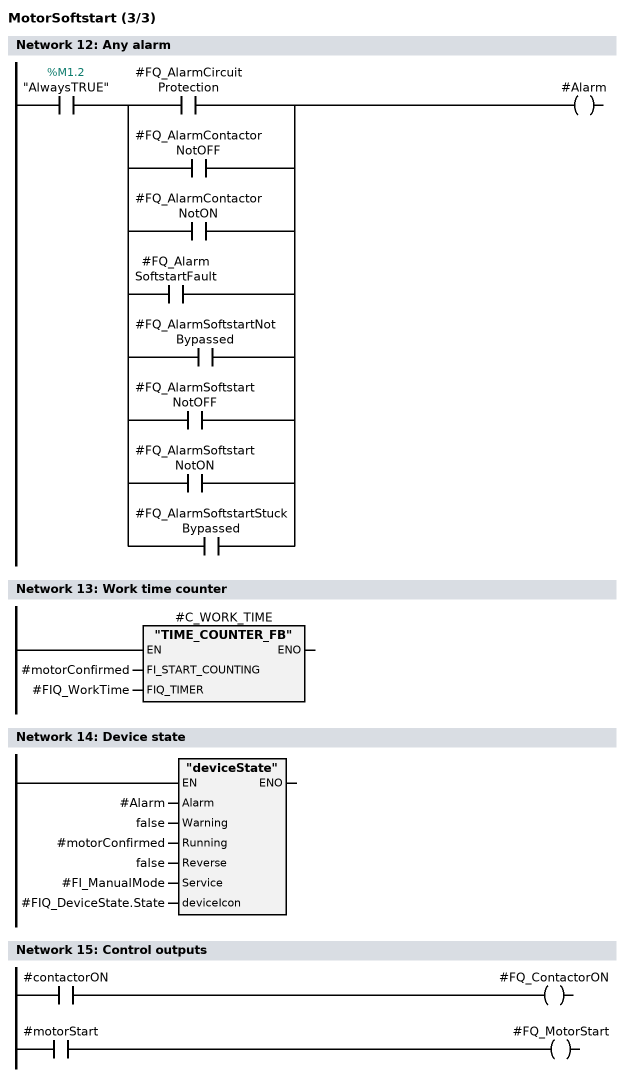
   RUNG wire#powerrail
      Contact( "AlwaysTRUE" )
      wire#w1
      Contact( #FQ_AlarmCircuitProtection )
      wire#w2
      Coil( #Alarm )
   END_RUNG
   RUNG wire#w1
      Contact( #FQ_AlarmContactorNotOFF )
   END_RUNG wire#w2
   RUNG wire#w1
      Contact( #FQ_AlarmContactorNotON )
   END_RUNG wire#w2
   RUNG wire#w1
      Contact( #FQ_AlarmSoftstartFault )
   END_RUNG wire#w2
   RUNG wire#w1
      Contact( #FQ_AlarmSoftstartNotBypassed )
   END_RUNG wire#w2
   RUNG wire#w1
      Contact( #FQ_AlarmSoftstartNotOFF )
   END_RUNG wire#w2
   RUNG wire#w1
      Contact( #FQ_AlarmSoftstartNotON )
   END_RUNG wire#w2
   RUNG wire#w1
      Contact( #FQ_AlarmSoftstartStuckBypassed )
   END_RUNG wire#w2
   // the same network as SCL:
   #Alarm := "AlwaysTRUE" AND (#FQ_AlarmCircuitProtection OR #FQ_AlarmContactorNotOFF OR #FQ_AlarmContactorNotON OR #FQ_AlarmSoftstartFault OR #FQ_AlarmSoftstartNotBypassed OR #FQ_AlarmSoftstartNotOFF OR #FQ_AlarmSoftstartNotON OR #FQ_AlarmSoftstartStuckBypassed);
END_REGION

REGION Network 13: Work time counter
   RUNG wire#powerrail
      #C_WORK_TIME(FI_START_COUNTING := #motorConfirmed, FIQ_TIMER := #FIQ_WorkTime)
   END_RUNG
   // the same network as SCL:
   #C_WORK_TIME(FI_START_COUNTING := #motorConfirmed, FIQ_TIMER := #FIQ_WorkTime);   // "TIME_COUNTER_FB"
END_REGION

REGION Network 14: Device state
   RUNG wire#powerrail
      "deviceState"(Alarm := #Alarm, Warning := false, Running := #motorConfirmed, Reverse := false, Service := #FI_ManualMode, deviceIcon := #FIQ_DeviceState.State)
   END_RUNG
   // the same network as SCL:
   "deviceState"(Alarm := #Alarm,
                 Warning := false,
                 Running := #motorConfirmed,
                 Reverse := false,
                 Service := #FI_ManualMode,
                 deviceIcon := #FIQ_DeviceState.State);
END_REGION

REGION Network 15: Control outputs
   RUNG wire#powerrail
      Contact( #contactorON )
      Coil( #FQ_ContactorON )
   END_RUNG
   RUNG wire#powerrail
      Contact( #motorStart )
      Coil( #FQ_MotorStart )
   END_RUNG
   // the same network as SCL:
   #FQ_ContactorON := #contactorON;
   #FQ_MotorStart := #motorStart;
END_REGION
END_FUNCTION_BLOCK

FUNCTION_BLOCK "TIME_COUNTER_FB"   // FB9000, LAD
{ S7_Optimized_Access := 'TRUE' }
// TIME COUNTER [S, M, H]
// stored: AutoNumber false, MemoryReserve 100, SetENOAutomatically false
   VAR_INPUT
      FI_START_COUNTING : Bool;
   END_VAR
   VAR_IN_OUT
      FIQ_TIMER : "UDT_WORK_CNT";
   END_VAR
   VAR
      E1 : Bool;
      E2 : Bool;
      RESET_CTU : Bool;
   END_VAR
   VAR_TEMP   // added for the SCL form of the ladder/FBD networks
      _w1 : Bool;
   END_VAR
BEGIN

REGION Network 1: COUNTERS INCREMENT
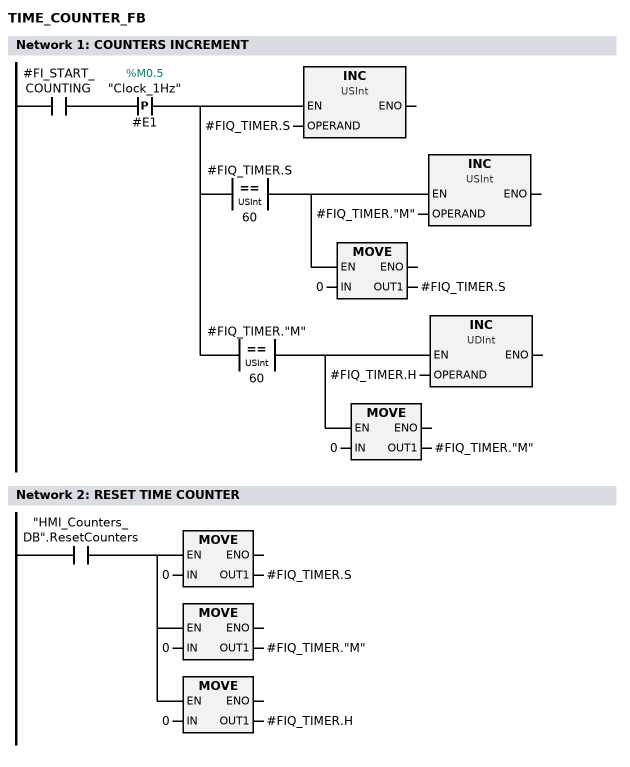
   RUNG wire#powerrail
      Contact( #FI_START_COUNTING )
      P_Contact(operand := "Clock_1Hz", bit := #E1)
      wire#w1
      { S7_Templates := "DestType := USInt" } Inc( #FIQ_TIMER.S )
   END_RUNG
   RUNG wire#w1
      { S7_Templates := "SrcType := USInt" } EQ_Contact(in1 := #FIQ_TIMER.S, in2 := 60)
      wire#w2
      { S7_Templates := "DestType := USInt" } Inc( #FIQ_TIMER."M" )
   END_RUNG
   RUNG wire#w2
      Move(in := 0, out1 => #FIQ_TIMER.S)
   END_RUNG
   RUNG wire#w1
      { S7_Templates := "SrcType := USInt" } EQ_Contact(in1 := #FIQ_TIMER."M", in2 := 60)
      wire#w3
      { S7_Templates := "DestType := UDInt" } Inc( #FIQ_TIMER.H )
   END_RUNG
   RUNG wire#w3
      Move(in := 0, out1 => #FIQ_TIMER."M")
   END_RUNG
   // the same network as SCL:
   #_w1 := #FI_START_COUNTING AND "Clock_1Hz" AND NOT #E1;   // rising edge of "Clock_1Hz"
   #E1 := "Clock_1Hz";
   IF #_w1 THEN #FIQ_TIMER.S := #FIQ_TIMER.S + 1; END_IF;
   IF #_w1 AND (#FIQ_TIMER.S = 60) THEN
       #FIQ_TIMER."M" := #FIQ_TIMER."M" + 1;
       #FIQ_TIMER.S := 0;
   END_IF;
   IF #_w1 AND (#FIQ_TIMER."M" = 60) THEN
       #FIQ_TIMER.H := #FIQ_TIMER.H + 1;
       #FIQ_TIMER."M" := 0;
   END_IF;
END_REGION

REGION Network 2: RESET TIME COUNTER
   RUNG wire#powerrail
      Contact( "HMI_Counters_DB".ResetCounters )
      wire#w1
      Move(in := 0, out1 => #FIQ_TIMER.S)
   END_RUNG
   RUNG wire#w1
      Move(in := 0, out1 => #FIQ_TIMER."M")
   END_RUNG
   RUNG wire#w1
      Move(in := 0, out1 => #FIQ_TIMER.H)
   END_RUNG
   // the same network as SCL:
   IF "HMI_Counters_DB".ResetCounters THEN
       #FIQ_TIMER.S := 0;
       #FIQ_TIMER."M" := 0;
       #FIQ_TIMER.H := 0;
   END_IF;
END_REGION
END_FUNCTION_BLOCK

DATA_BLOCK "FB_Sensores_DB"   // DB2
// stored: InstanceOfName FB_Sensores, InstanceOfType FB
"FB_Sensores"
BEGIN
END_DATA_BLOCK

DATA_BLOCK "HMI_Settings_DB"   // DB703
{ S7_Optimized_Access := 'TRUE'; DB_Accessible_From_OPC_UA := 'FALSE' }
// stored: AutoNumber false, DBAccessibleFromOPCUA false, DBAccessibleFromWebserver false, InstanceOfName UDT_Settings, InstanceOfType UDT
"UDT_Settings"
BEGIN
END_DATA_BLOCK
